// LS Electric XG5000 project: 0131 인버터
// PLC LSPLC

PROGRAM NewProgram (task: 스캔 프로그램)

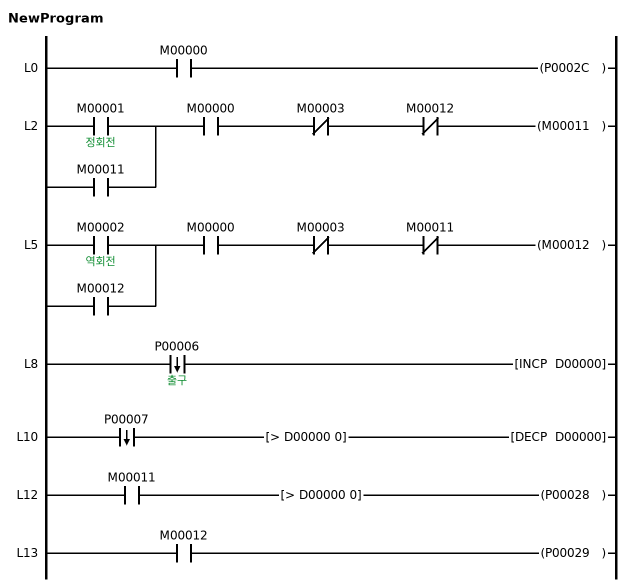
; L0
LOAD      M00000
OUT       P0002C
; L2
LOAD      M00001	// 정회전
OR        M00011
AND       M00000
AND NOT   M00003
AND NOT   M00012
OUT       M00011
; L5
LOAD      M00002	// 역회전
OR        M00012
AND       M00000
AND NOT   M00003
AND NOT   M00011
OUT       M00012
; L8
LOADN     P00006	// 출구
INCP      D00000
; L10
LOADN     P00007
AND>      D00000 0
DECP      D00000
; L12
LOAD      M00011
AND>      D00000 0
OUT       P00028
; L13
LOAD      M00012
OUT       P00029